FUNCTION SIGN_R : BOOL
VAR_INPUT
	in : REAL;
END_VAR


(*
version 1.4	10. mar. 2009
programmer 	hugo
tested by		tobias

this function return true if the real input is negative

*)

SIGN_R := in < 0.0;


(* revision history
hm 19.1.2007	rev 1.1
	changed method of function for better compatibility to other systems

hm	1.12.2007	rev 1.2
	changed code to improve performance

hm	14. jun. 2008	rev 1.3
	improved performace

hm 10. mar. 2009	rev 1.4
	real constants updated to new systax using dot																																																																																																																																																																																																																																																																																																																																																																																																																																																																																																																																																																																																																																																																																																																																																																																																																																																																																																																																																																																																																																																											

*)

END_FUNCTION

(* stored: Version 1.1.0.1, ProductVersion 3.1.4022.7
   POU SIGN_R: Id {b0e16301-eeeb-4a67-9ebb-085681f398a6}, SpecialFunc None *)
